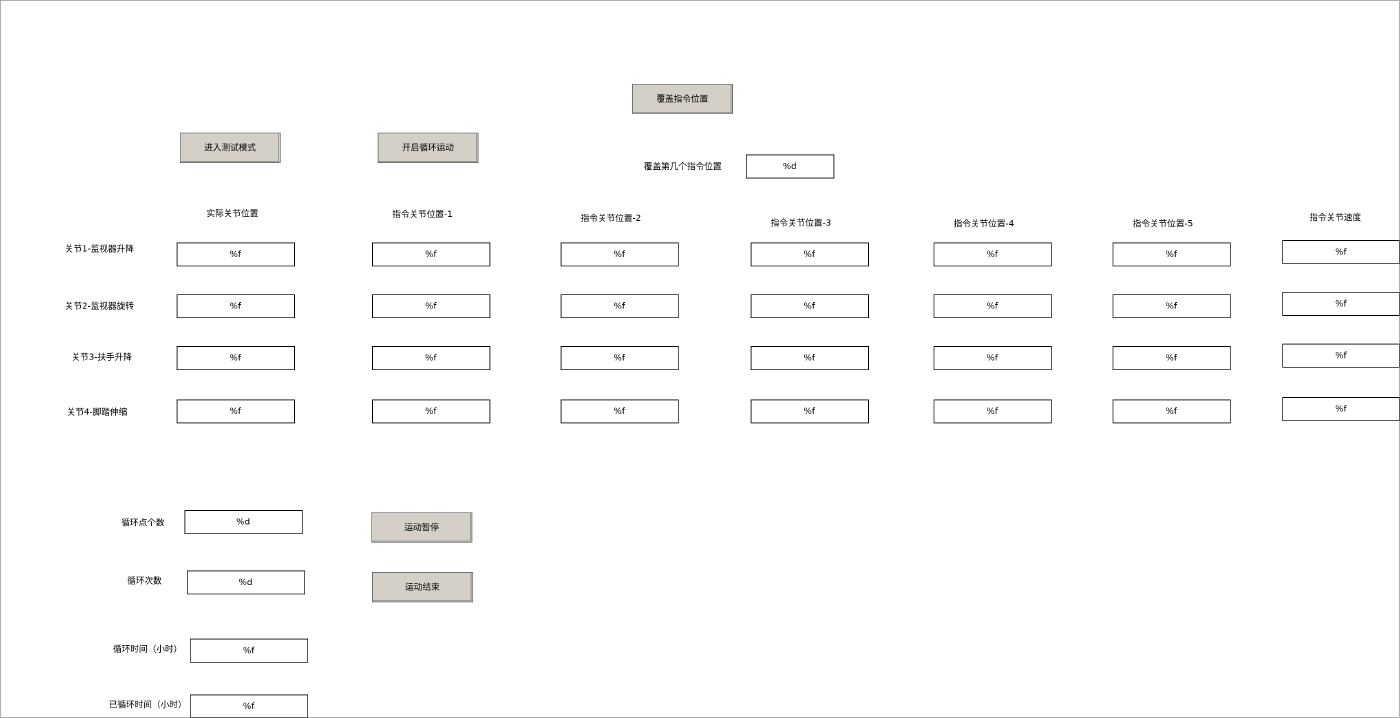
VISUALIZATION cycle_car  // 1783x915
    Label (221,257 150x30), "实际关节位置"
    Rectangle (225,309 150x30), "%f", text variable: g_cycleTest.m_carJntPos[1]
    Label (463,258 150x30), "指令关节位置-1"
    Button (229,169 128x38), "进入测试模式", colour toggle: g_cycleTest.m_carEnterCycleTest
        toggle g_cycleTest.m_carEnterCycleTest
    Button (481,169 128x38), "开启循环运动", colour toggle: g_cycleTest.m_startMotionCar
        toggle g_cycleTest.m_startMotionCar
    Rectangle (225,375 150x30), "%f", text variable: g_cycleTest.m_carJntPos[2]
    Rectangle (225,441 150x30), "%f", text variable: g_cycleTest.m_carJntPos[3]
    Rectangle (225,509 150x30), "%f", text variable: g_cycleTest.m_carJntPos[4]
    Rectangle (474,309 150x30), "%f", text variable: g_cycleTest.m_targetJntPosCar[1][1]
        OnMouseClick: write the text variable via Default
    Rectangle (474,375 150x30), "%f", text variable: g_cycleTest.m_targetJntPosCar[1][2]
        OnMouseClick: write the text variable via Default
    Rectangle (474,441 150x30), "%f", text variable: g_cycleTest.m_targetJntPosCar[1][3]
        OnMouseClick: write the text variable via Default
    Rectangle (474,509 150x30), "%f", text variable: g_cycleTest.m_targetJntPosCar[1][4]
        OnMouseClick: write the text variable via Default
    Label (703,263 150x30), "指令关节位置-2"
    Rectangle (714,309 150x30), "%f", text variable: g_cycleTest.m_targetJntPosCar[2][1]
        OnMouseClick: write the text variable via Default
    Rectangle (714,375 150x30), "%f", text variable: g_cycleTest.m_targetJntPosCar[2][2]
        OnMouseClick: write the text variable via Default
    Rectangle (714,441 150x30), "%f", text variable: g_cycleTest.m_targetJntPosCar[2][3]
        OnMouseClick: write the text variable via Default
    Rectangle (714,509 150x30), "%f", text variable: g_cycleTest.m_targetJntPosCar[2][4]
        OnMouseClick: write the text variable via Default
    Label (945,269 150x30), "指令关节位置-3"
    Rectangle (956,309 150x30), "%f", text variable: g_cycleTest.m_targetJntPosCar[3][1]
        OnMouseClick: write the text variable via Default
    Rectangle (956,375 150x30), "%f", text variable: g_cycleTest.m_targetJntPosCar[3][2]
        OnMouseClick: write the text variable via Default
    Rectangle (956,441 150x30), "%f", text variable: g_cycleTest.m_targetJntPosCar[3][3]
        OnMouseClick: write the text variable via Default
    Rectangle (956,509 150x30), "%f", text variable: g_cycleTest.m_targetJntPosCar[3][4]
        OnMouseClick: write the text variable via Default
    Label (1178,270 150x30), "指令关节位置-4"
    Rectangle (1189,309 150x30), "%f", text variable: g_cycleTest.m_targetJntPosCar[4][1]
        OnMouseClick: write the text variable via Default
    Rectangle (1189,375 150x30), "%f", text variable: g_cycleTest.m_targetJntPosCar[4][2]
        OnMouseClick: write the text variable via Default
    Rectangle (1189,441 150x30), "%f", text variable: g_cycleTest.m_targetJntPosCar[4][3]
        OnMouseClick: write the text variable via Default
    Rectangle (1189,509 150x30), "%f", text variable: g_cycleTest.m_targetJntPosCar[4][4]
        OnMouseClick: write the text variable via Default
    Label (1406,270 150x30), "指令关节位置-5"
    Rectangle (1417,309 150x30), "%f", text variable: g_cycleTest.m_targetJntPosCar[5][1]
        OnMouseClick: write the text variable via Default
    Rectangle (1417,375 150x30), "%f", text variable: g_cycleTest.m_targetJntPosCar[5][2]
        OnMouseClick: write the text variable via Default
    Rectangle (1417,441 150x30), "%f", text variable: g_cycleTest.m_targetJntPosCar[5][3]
        OnMouseClick: write the text variable via Default
    Rectangle (1417,509 150x30), "%f", text variable: g_cycleTest.m_targetJntPosCar[5][4]
        OnMouseClick: write the text variable via Default
    Label (107,651 150x30), "循环点个数"
    Rectangle (235,650 150x30), "%d", text variable: g_cycleTest.m_pointSumCar
        OnMouseClick: write the text variable via Default
    Rectangle (238,727 150x30), "%d", text variable: g_cycleTest.m_curCycleNumCar
        OnMouseClick: write the text variable via Default
    Label (109,725 150x30), "循环次数"
    Button (473,653 128x38), "运动暂停", colour toggle: g_cycleTest.m_pauseCar
        toggle g_cycleTest.m_pauseCar
    Button (474,729 128x38), "运动结束", colour toggle: g_cycleTest.m_finishCar
        tap g_cycleTest.m_finishCar
    Label (54,303 145x28), "关节1-监视器升降"
    Label (54,376 145x28), "关节2-监视器旋转"
    Label (57,441 145x28), "关节3-扶手升降"
    Label (51,511 145x28), "关节4-脚踏伸缩"
    Rectangle (242,814 150x30), "%f", text variable: g_cycleTest.m_tgtCycleTimeCar
        OnMouseClick: write the text variable via Default
    Label (113,812 150x30), "循环时间（小时）"
    Rectangle (242,885 150x30), "%f", text variable: g_cycleTest.m_curCycleTimeCar
        OnMouseClick: write the text variable via Default
    Label (113,883 150x30), "已循环时间（小时）"
    Button (805,107 128x38), "覆盖指令位置", colour toggle: g_cycleTest.m_coverCmdPosCar
        tap g_cycleTest.m_coverCmdPosCar
    Rectangle (950,197 112x30), "%d", text variable: g_cycleTest.m_pntIdForCoverCmdCar
        OnMouseClick: write the text variable via Default
    Label (797,198 145x28), "覆盖第几个指令位置"
    Label (1628,263 145x28), "指令关节速度"
    Rectangle (1633,306 150x30), "%f", text variable: g_cycleTest.m_targetJntVelCar[1]
        OnMouseClick: write the text variable via Default
    Rectangle (1633,372 150x30), "%f", text variable: g_cycleTest.m_targetJntVelCar[2]
        OnMouseClick: write the text variable via Default
    Rectangle (1633,438 150x30), "%f", text variable: g_cycleTest.m_targetJntVelCar[3]
        OnMouseClick: write the text variable via Default
    Rectangle (1633,506 150x30), "%f", text variable: g_cycleTest.m_targetJntVelCar[4]
        OnMouseClick: write the text variable via Default
END_VISUALIZATION

(* stored: Version 1.1.0.1, ProductVersion 3.1.4024.11
   Visu cycle_car: Id {287e4461-315c-48a4-a0e8-9f133537216e} *)
